PROGRAM PRG_Turntable
VAR
	Turntable : CTURNTABLE;

	
	SaleCajaA : BOOL;
	SaleCajaV : BOOL;
	SaleCajaM : BOOL;
	
	iCajaProcesando : INT;
	
	tFTrigDiffuseSensor	: F_TRIG;
	tFTrigEmitterA: F_TRIG;
	tFTrigEmitterV: F_TRIG;
	tFTrigEmitterM: F_TRIG;
END_VAR

tFTrigDiffuseSensor(CLK:= GVL_ProcesoPalet.bDiffuseSensorSalida);
tFTrigEmitterA(CLK:= GVL_ProcesoPalet.iLightArrayEmitterA);
tFTrigEmitterV(CLK:= GVL_ProcesoPalet.iLightArrayEmitterV);
tFTrigEmitterM(CLK:= GVL_ProcesoPalet.iLightArrayEmitterM);

CASE Turntable OF
	
	CTURNTABLE_ESPERA:
	(* Dependiendo de las detecciones de los sensores, se activarám según qué líneas*)
	
	IF POU_PickAndPlace.CajaLlenaA THEN
		SaleCajaA := TRUE;
		GVL_ProcesoPalet.sRollerConveyor.bRollerAzul1 := TRUE;
		GVL_ProcesoPalet.sRollerConveyor.bCurvedRollerAzul1 := TRUE;
		
		IF tFTrigEmitterA.Q THEN
			Turntable := CTURNTABLE_FILTROPRIORIDAD;
			iCajaProcesando := iCajaProcesando + 1;
		END_IF
	END_IF
	
	IF POU_PickAndPlace.CajaLlenaV THEN
		SaleCajaV := TRUE;
		GVL_ProcesoPalet.sRollerConveyor.bRollerVerde1 := TRUE;
		Turntable := CTURNTABLE_FILTROPRIORIDAD;
		
		IF tFTrigEmitterV.Q THEN
			Turntable := CTURNTABLE_FILTROPRIORIDAD;
			iCajaProcesando := iCajaProcesando + 1;
		END_IF
	END_IF
	
	IF POU_PickAndPlace.CajaLlenaM THEN
		SaleCajaM := TRUE;
		GVL_ProcesoPalet.sRollerConveyor.bRollerMetal1 := TRUE;
		GVL_ProcesoPalet.sRollerConveyor.bCurvedRollerMetal1 := TRUE;
		
		IF tFTrigEmitterM.Q THEN
			Turntable := CTURNTABLE_FILTROPRIORIDAD;
			iCajaProcesando := iCajaProcesando + 1;
		END_IF
	END_IF

	
	CTURNTABLE_FILTROPRIORIDAD:
	(* Dependiendo de las detecciones de los sensores, se girará a una posición u otra*)
	
	IF GVL_ProcesoPalet.bDiffuseSensorPaletA THEN
		SaleCajaA := FALSE;
		GVL_ProcesoPalet.sRollerConveyor.bCurvedRollerAzul1 := FALSE;
		TURNTABLE := CTURNTABLE_CARGAAZUL;
	END_IF
	
	IF GVL_ProcesoPalet.bDiffuseSensorPaletV THEN
		GVL_ProcesoPalet.sRollerConveyor.bRollerVerde1 := FALSE;
		TURNTABLE := CTURNTABLE_CARGAVERDE;
	END_IF
	
	IF GVL_ProcesoPalet.bDiffuseSensorPaletM THEN
		GVL_ProcesoPalet.sRollerConveyor.bCurvedRollerMetal1 := FALSE;
		TURNTABLE := CTURNTABLE_CARGAMETAL;
	END_IF
		
	
	CTURNTABLE_CARGAAZUL:
	(* Proceso de carga para la caja azul *)
	
	GVL_ProcesoPalet.sTurnTable.Turn := TRUE;
	GVL_ProcesoPalet.sTurnTable.RollPositivo := TRUE;
	
	IF GVL_ProcesoPalet.sTurnTable.Limit90 THEN
		TURNTABLE := CTURNTABLE_DESCARGAAZUL;
	END_IF	
	
	
	CTURNTABLE_DESCARGAAZUL:
	(* Proceso de descarga para la caja azul *)
	
	GVL_ProcesoPalet.sRollerConveyor.bCurvedRollerAzul1 := TRUE;
	IF GVL_ProcesoPalet.sTurnTable.FrontLimit THEN
		GVL_ProcesoPalet.sTurnTable.RollPositivo := FALSE;
		GVL_ProcesoPalet.sTurnTable.Turn := FALSE;
	END_IF
	
	IF GVL_ProcesoPalet.sTurnTable.Limit0 THEN
		GVL_ProcesoPalet.sTurnTable.RollPositivo := TRUE;
		TURNTABLE := CTURNTABLE_SALIDA;
	END_IF
	
	
	CTURNTABLE_CARGAVERDE:
	(* Proceso de carga para la caja verde *)
	
	GVL_ProcesoPalet.sTurnTable.Turn := FALSE;
	IF GVL_ProcesoPalet.sTurnTable.Limit0 THEN
		GVL_ProcesoPalet.sRollerConveyor.bRollerVerde1 := TRUE;
		GVL_ProcesoPalet.sTurnTable.RollPositivo := TRUE;
		TURNTABLE := CTURNTABLE_SALIDA;
	END_IF
	
	
	CTURNTABLE_CARGAMETAL:
	(* Proceso de carga para la caja azul *)
	
	GVL_ProcesoPalet.sTurnTable.Turn := TRUE;
	GVL_ProcesoPalet.sTurnTable.RollNegativo := TRUE;
	
	IF GVL_ProcesoPalet.sTurnTable.Limit90 THEN
		TURNTABLE := CTURNTABLE_DESCARGAMETAL;
	END_IF	
	
	
	CTURNTABLE_DESCARGAMETAL:
	(* Proceso de descarga para la caja azul *)
	
	GVL_ProcesoPalet.sRollerConveyor.bCurvedRollerMetal1 := TRUE;
	IF GVL_ProcesoPalet.sTurnTable.BackLimit THEN
		GVL_ProcesoPalet.sTurnTable.RollNegativo := FALSE;
		GVL_ProcesoPalet.sTurnTable.Turn := FALSE;
	END_IF
	
	IF GVL_ProcesoPalet.sTurnTable.Limit0 THEN
		GVL_ProcesoPalet.sTurnTable.RollPositivo := TRUE;
		TURNTABLE := CTURNTABLE_SALIDA;
	END_IF
	
	
	CTURNTABLE_SALIDA:

	IF tFTrigDiffuseSensor.Q THEN
		TURNTABLE := CTURNTABLE_ESPERA;
		GVL_ProcesoPalet.sTurnTable.RollPositivo := FALSE;
	END_IF
	
END_CASE

END_PROGRAM

(* stored: Version 1.1.0.1, ProductVersion 3.1.4024.12
   POU PRG_Turntable: Id {4632a491-dbef-4586-9e55-e4a069d82d54}, SpecialFunc None *)
